	      ELSE
	        // Fehlerwiederholauftrag ??                   
	        IF #siErrorCount = #siMaxErrCount THEN
	          
	          // Wiederholungsauftrag wieder zurücknehmen
	          #sbWrStart2 := False;
	          #sbRdStart2 := False;
	          #sbWrite := False;
	          
	          //Fehlerzähler zurücksetzen
	          #siErrorCount := 0;
	          
	          
	          // Fehler ausgeben 
	          #sbError := #sbRdError;
	          
	          // nix tun bis Zähler überläuft
	        ELSE
	          #siErrorCount := #siErrorCount + 1;
	        END_IF;
	      END_IF;
	      
	      // Fehler : die Auftragsreferenz der Antwort übertimmt nicht mit der Auftragsreferenz der Anfrage überein
	    ELSIF NOT (#siReqRef = BYTE_TO_INT(#sxRespParaMulti.sxHeader.syReqRef)) AND NOT #sbRdBusy AND #pbValidSFB THEN
	      #siErrorId := 1;
	      #sbError := True;
	      #sbDone := False;
	      
	      // Wiederholungsauftrag wieder zurücknehmen
	      #sbWrStart2 := False;
	      #sbRdStart2 := False;
	      #sbWrite := False;
	      
	      // Fehler : falsche Auftragskennung zurück erhalten    
	    ELSIF NOT (#sxRespParaMulti.sxHeader.syReqId = B#16#82 OR #sxRespParaMulti.sxHeader.syReqId = B#16#02) AND
	      NOT #sbRdBusy AND #pbValidSFB THEN
	      #siErrorId := 1;
	      #sbError := True;
	      #sbDone := False;
	      
	      // Wiederholungsauftrag wieder zurücknehmen
	      #sbWrStart2 := False;
	      #sbRdStart2 := False;
	      #sbWrite := False;
	      
	      // Fehler : die angeforderte Anzahl Parameter entspricht nicht der übermittelten Anzahl Parameter überein
	    ELSIF NOT (#sxRespParaMulti.sxHeader.syParaNo = B#16#01) AND NOT #sbRdBusy AND #pbValidSFB THEN
	      #siErrorId := 1;
	      #sbError := True;
	      #sbDone := False;
	      
	      // Wiederholungsauftrag wieder zurücknehmen
	      #sbWrStart2 := False;
	      #sbRdStart2 := False;
	      #sbWrite := False;
	      
	      // Fehler : die Achse entspricht nicht der übergebenen Achse
	    ELSIF NOT (#syAxisNo = #sxRespParaMulti.sxHeader.syAxisNo) AND NOT #sbRdBusy AND #pbValidSFB THEN
	      #siErrorId := 1;
	      #sbError := True;
	      #sbDone := False;
	      
	      // Wiederholungsauftrag wieder zurücknehmen
	      #sbWrStart2 := False;
	      #sbRdStart2 := False;
	      #sbWrite := False;
	      
	      // kein Fehler beim LESEN AZYKLISCH und Auftrag fertig 
	    ELSIF NOT #sbRdBusy AND #pbValidSFB THEN
	      
	      // 2. Teilauftrag "Parameter schreiben bzw. ändern" negative Rückmeldung erhalten 
	      IF #sxRespParaMulti.sxHeader.syReqId = B#16#82 THEN
	        
	        // die angefragten Parameter auswerten und im Puffer abspeichern
	        // Format des Parameters auswerten, bei Format = Error Fehler auswerten 
	        IF (BYTE_TO_INT(#sxRespParaMulti.sxData[1]) = 68) THEN
	          
	          // Fehlerwert ermitteln und abspeichern 
	          // Format = Word, zwei Bytes zu übermitteltem Parameterwert zusammenfassen
	          #pwWordHigh := SHL(IN := BYTE_TO_WORD(#sxRespParaMulti.sxData[3]), N := 8);
	          #pwWordLow := BYTE_TO_WORD(#sxRespParaMulti.sxData[4]);
	          #pwWord1 := #pwWordHigh XOR #pwWordLow;
	            
	          #sbError := True;
	            
	          // ermittelte Fehlernummer im Puffer zurücksetzen
	          #ErrorNo := W#16#00;
	          
	          #ErrorNo := #pwWord1;
	          
	          // Die Fehlerhaftigkeit des erkannten Parameter in der Fehlernummer eintragen   
	          #swParaError := #swParaError OR W#16#01;
	          
	        ELSE
	          
	          // Die Fehlerhaftigkeit des erkannten Parameter in der Fehlernummer löschen   
	          #swParaError := #swParaError AND W#16#FFFE;
	          
	          // ermittelte Fehlernummer im Puffer zurücksetzen
	          #ErrorNo := W#16#00;
	        END_IF;
	      END_IF; // 2. Teilauftrag "Parameter schreiben bzw. ändern" negative Rückmeldung erhalten
	      
	      // Fehlerkennung zurücknehmen
	      IF (#siErrorId = 3) OR (#siErrorId = 1) THEN
	        #siErrorId := 0;
	        #sbError := False;
	      END_IF;
	      
	      #DiagId := W#16#00;
	      
	      // 2. Teilauftrag "Parameter schreiben bzw. ändern" ist abgeschlossen
	      #sbRdStart2 := False;
	      #sbWrite := False;
	      
	    END_IF; // kein Fehler beim LESEN AZYKLISCH und Auftrag fertig 
	  END_IF; // vom 2. Teilauftrag "Parameter schreiben bzw. ändern" die Antwort abwarten und dann auswerten 
	END_IF; // Auftrag "Parameter schreiben" wurde ausgelöst
	
	#pdDWordHigh := SHL(IN := INT_TO_DWORD(#siErrorId), N := 16);
	#pdDWordLow := WORD_TO_DWORD(#swParaError);
	
	// ermittelter Parameterwert eintragen (Word)
	#ErrorId := #pdDWordHigh XOR #pdDWordLow;
	
	// Initialisierung von Ausgängen
	#Busy := #sbBusy;
	#Error := #sbError;
	#Format := #syFormat;
	// Änderung wegen verhalten von Ready  
	#Done := #sbDone;
	// Prüfen, ob Auftrag abgeschlossen ist
	IF ((#Error OR #Done) AND NOT #sbReady) THEN
	  #Ready := True;
	  #sbReady := True;
	ELSE
	  #Ready := False;
	END_IF;
	
	
END_FUNCTION_BLOCK

FUNCTION_BLOCK "SINA_SPEED"
TITLE = 'Speed Control with SINAMICS and S7'
{ S7_Optimized_Access := 'TRUE' }
AUTHOR : DRVDPS7
FAMILY : DRIVES
NAME : SINA_SPD
VERSION : 5.1
//Copyright (C) Siemens AG 2012. All Rights Reserved. Confidential
//-------------------------------------------------------------------------------------- 
//SINA_SPEED: Drehzahlregelung mit dem Antriebsbaustein SINAMICS S120/G120 <-> S7-1200
//------------------------------------------------------------------------------------- Ersteller: Siemens AG Erlangen A&D MC PM   Datum:  07.07.10        Vers.:2.1
//Änderung:  J.B. Typical Team                       07.12.12              2.2
//    Umsetzung in SCL / TIA 
//Änderung:  J.B. Typical Team                       29.04.13              2.3
//    1. "Q" an den AusgÃ¤nge entfernen
//    2. Neuer Ausgang PwrInhibit
//Änderung:  J.B. Typical Team                       28.06.13              2.4
//    Ã„nderung HW-Zugriff Ã¼ber LOG2MOD
//     
//Änderung:  J.B. Typical Team                       18.07.13              2.5
//    Ã„nderung HW-Zugriff Ã¼ber zwei HW-EingÃ¤nge
//
//Änderung:  J.B. Typical Team                       17.07.14              3.0
//    Optimmierung
//
//Änderung:  J.B. Typical Team                       30.07.14              4.0
//    Festlegung auf einheitlicher neuer Version 4.0
//
//Änderung:  P.Z. Typical Team                       03.12.15              4.1
//    Schnittstelle an Programmierleitfadeb TIA-Potal angepasst
//    zusÃ¤tzlicher Eingang "ConfigAxis" fÃ¼r STW-Bits
//
//Änderung:  G.F. Typical Team                       01.03.16              4.2
//    Sollwert auf INT - Grenzen begrenzt
//Änderung:  F.G. Typical Team                       13.09.16              4.3
//    Ausgabewerte am Ausgang "Status" angepasst 
//
//Änderung:  G.F. Typical Team                       11.01.17              5.0
//    - Festlegung auf einheitlicher neuer Version 5.0 
//
//Änderung:  G.F. Typical Team                       03.05.18              5.1
//    - Alle Bits des Eingang ConfigAxis auf STW1 aufgelegt 
//
//Bibliothek V7
//Funktion: Drehzahlregelung mit dem Antriebsbaustein SINAMICS S120/G120 <-> S7-1200
//********************************************************************************************************************************************************
//************************************************************************FB283***************************************************************************
//********************************************************************************************************************************************************
   VAR_INPUT 
      EnableAxis : Bool := 0;   // 0-->1; 1 = Enable the drive (OFF2 / OFF 3 are 1 in default status) (OFF1 = 0-->1)
      AckError : Bool := 0;   // 1 = Acknowledge drive error
      SpeedSp : Real := 0.0;   // Speed standardises with the standardisation factor
      RefSpeed : Real := 0.0;   // Standardisation factor of speed
      ConfigAxis : Word := 16#003F;   // binary programmed input to control all functions in the telegram without its own function block input
      HWIDSTW : HW_IO := 0;   // Hardware Identifer set point slot
      HWIDZSW : HW_IO := 0;   // Hardware Identifer actual value slot
   END_VAR

   VAR_OUTPUT 
      AxisEnabled : Bool := 0;   // 1 = Drive is enabled
      Lockout : Bool := 0;   // 1 = Drive lockout active
      ActVelocity : Real := 0.0;   // Actual in [U/min]
      Error : Bool := 0;   // 1 = Error  (FB and Infeed)
      Status : Word := 0;   // Status output (7002 = FB in operation; 8xxx = error description  - read the manual)
      DiagId : Word := 16#0000;   // Error codes of the cyclic system funtion blocks DPWR / DPRD_DAT
   END_VAR

   VAR 
      sxSendBuf : Struct   // Send buffer
         STW1 : Word := WORD#16#0000;   // STW1sxSTW1     : STRUCT            Bit08       : BOOL:=False;              // ST-Wort-1 Bit 08 --> Reserve            Bit09       : BOOL:=False;              // ST-Wort-1 Bit 09 --> Reserve            Bit10       : BOOL:=True;               // ST-Wort-1 Bit 10 --> FÃ¼hrung durch PLC            Dir         : BOOL:=False;              // ST-Wort-1 Bit 11 --> Direction            Bit12       : BOOL:=False;              // ST-Wort-1 Bit 12 --> Haltebremse unbedingt Ã¶ffnen            Bit13       : BOOL:=False;              // ST-Wort-1 Bit 13 --> Motorpotenziometer Sollwert hÃ¶her            Bit14       : BOOL:=False;              // ST-Wort-1 Bit 14 --> Motorpotenziometer Sollwert tiefer            Bit15       : BOOL:=False;              // ST-Wort-1 Bit 15 --> Reserviert            Off1        : BOOL:=False;              // ST-Wort-1 Bit 00 --> OFF1/ON (flanks acceptance)            Off2        : BOOL:=True;               // ST-Wort-1 Bit 01 --> OFF2/ON (enable possible)            Off3        : BOOL:=True;               // ST-Wort-1 Bit 02 --> OFF3/ON (enable possible)            InvEn       : BOOL:=True;               // ST-Wort-1 Bit 03 --> Enable controller            RampEn      : BOOL:=True;               // ST-Wort-1 Bit 04 --> Ramp enable            RampOn      : BOOL:=True;               // ST-Wort-1 Bit 05 --> Ramp On            SpEn        : BOOL:=True;               // ST-Wort-1 Bit 06 --> Speed set point enable            AckFlt      : BOOL:=False;              // ST-Wort-1 Bit 07 --> Acknowledge fault         END_STRUCT;
         Velocity : Word := WORD#16#0000;   // Setpoint of velocity
      END_STRUCT;
      sxRecvBuf : Struct   // Receive buffer
         ZSW1 : Word := WORD#16#0000;   // ZSW1sxZSW1     : STRUCT            SpDev       : BOOL:=False;              // ZSW-Wort-1 = Schleppfehler im Toleranzbereich            Pcd         : BOOL:=False;              // ZSW-Wort-1 = PZD-FÃ¼hrung erreicht            Comp        : BOOL:=False;              // ZSW-Wort-1 = Zielposition erreicht            CurLim      : BOOL:=False;              // ZSW-Wort-1 = Referenzpunkt gesetzt            Brake       : BOOL:=False;              // ZSW-Wort-1 = Haltebremse Ã¶ffnen            Motover     : BOOL:=False;              // ZSW-Wort-1 = keine Warnung Ãœbertemperatur Motor            Dir         : BOOL:=False;              // ZSW-Wort-1 = Direction            Invover     : BOOL:=False;              // ZSW-Wort-1 = keine Warnung thermische Ãœberlast Leistungsteil            Rts         : BOOL:=False;              // ZSW-Wort-1 = Ready to power up / to start            Rdy         : BOOL:=False;              // ZSW-Wort-1 = Ready to operate            IOp         : BOOL:=False;              // ZSW-Wort-1 = In operation (operation enabled)            Fault       : BOOL:=False;              // ZSW-Wort-1 = Fault present            NoOff2      : BOOL:=False;              // ZSW-Wort-1 = OFF2 inactive            NoOff3      : BOOL:=False;              // ZSW-Wort-1 = OFF3 inactive            Inhibit     : BOOL:=False;              // ZSW-Wort-1 = Power ON inhibit active             Alarm       : BOOL:=False;              // ZSW-Wort-1 = Alarm / Warning present                     END_STRUCT;
         Velocity : Word := WORD#16#0000;   // Feedback of velocity
      END_STRUCT;
   END_VAR

   VAR_TEMP 
      piRetSFC : Int;   // Status for fault analysis
      piCount : Int;   // Freely available counter variable 3
      prVelocity : Real;   // velocity
      pdRecvBuf : DWord;   // Buffer of Recv-Value
      pdSendBuf : DWord;   // Buffer of Send-Value
      phLAddr : HW_IO;   // Start addr from the I/O process image area of mod (DEC) for DPWR_DAT/DPRD_DAT
      swSendBuf : Array[0..1] of Word;   // Sendepuffer
      swRecvBuf : Array[0..1] of Word;   // Empfangspuffer         Static variables
   END_VAR


BEGIN
	
	//=============================================================================
	//SIEMENS AG
	//(c)Copyright 2017 All Rights Reserved
	//-----------------------------------------------------------------------------
	// Library: DriveLib
	// Tested with: S7-1516-3 PN/DP V1.8
	// Engineering: TIA Portal V14
	// Restrictions: -
	// Requirements: S7-1200 / S7-1500
	// Functionality: cyclic communication between a SINAMICS a PLC.
	//                If in HWConfig Std.TLG 1 is projected 2 PZD-words are exchanged
	//                in every bus cycle.
	//                The parametrisation of these words is described in the manual of the
	//                SINAMICS
	//=============================================================================
	
	// Schreibdaten zusammenstellen
	// Steuerword aufbereiten
	
	#sxSendBuf.STW1.%X0 := #EnableAxis;
	#sxSendBuf.STW1.%X1 := #ConfigAxis.%X0;
	#sxSendBuf.STW1.%X2 := #ConfigAxis.%X1;
	#sxSendBuf.STW1.%X3 := #ConfigAxis.%X2;
	#sxSendBuf.STW1.%X4 := #ConfigAxis.%X3;
	#sxSendBuf.STW1.%X5 := #ConfigAxis.%X4;
	#sxSendBuf.STW1.%X6 := #ConfigAxis.%X5;
	#sxSendBuf.STW1.%X7 := #AckError;
	#sxSendBuf.STW1.%X8 := #ConfigAxis.%X10;
	#sxSendBuf.STW1.%X9 := #ConfigAxis.%X11;
	#sxSendBuf.STW1.%X10 := TRUE;
	#sxSendBuf.STW1.%X11 := #ConfigAxis.%X6;
	#sxSendBuf.STW1.%X12 := #ConfigAxis.%X7;
	#sxSendBuf.STW1.%X13 := #ConfigAxis.%X8;
	#sxSendBuf.STW1.%X14 := #ConfigAxis.%X9;
	#sxSendBuf.STW1.%X15 := #ConfigAxis.%X12;
	
	// Geschwindigkeit
	IF #RefSpeed <> 0 THEN
	  #prVelocity := #SpeedSp * (16384.0 / #RefSpeed);
	  // Limit REAL - Variable to INT - Limits
	  IF #prVelocity > 32767 THEN
	    #prVelocity := 32767;
	  ELSIF #prVelocity < -32768 THEN
	    #prVelocity := -32768;
	  ELSE
	    ; // not needed
	  END_IF;
	  #sxSendBuf.Velocity := INT_TO_WORD(REAL_TO_INT(#prVelocity));
	  
	ELSE
	  #sxSendBuf.Velocity := W#16#0;
	END_IF;
	#swSendBuf[0] := #sxSendBuf.STW1;
	#swSendBuf[1] := #sxSendBuf.Velocity;
	
	//Prozessdaten zur Signalbaugruppe schreiben
	#piRetSFC := DPWR_DAT(LADDR := #HWIDSTW,
	                      RECORD := #swSendBuf);
	
	// Fehler der RÃ¼ckmeldung ausgeben
	#DiagId := INT_TO_WORD(#piRetSFC);
	
	//kein Fehler beim Schreiben
	IF #piRetSFC = 0 THEN
	  
	  //kein Fehler beim Schreiben
	  IF #piRetSFC = 0 THEN
	    
	    //Prozessdaten von der Signalbaugruppe lesen
	    #piRetSFC := DPRD_DAT(LADDR := #HWIDZSW,
	                          RECORD => #swRecvBuf);
	    
	    // Fehler der RÃ¼ckmeldung ausgeben
	    #DiagId := INT_TO_WORD(#piRetSFC);
	  END_IF;
	  
	  //Fehler beim Lesen (Profibus-Kommunikation unterbrochen)
	  IF #piRetSFC <> 0 THEN
	    
	    // Fehler
	    #Error := TRUE;
	    #Status := 16#8600;
	    
	    // Zustandsworte lÃ¶schen
	    #sxRecvBuf.ZSW1.%X8 := 0;
	    #sxRecvBuf.ZSW1.%X9 := 0;
	    #sxRecvBuf.ZSW1.%X10 := 0;
	    #sxRecvBuf.ZSW1.%X11 := 0;
	    #sxRecvBuf.ZSW1.%X12 := 0;
	    #sxRecvBuf.ZSW1.%X13 := 0;
	    #sxRecvBuf.ZSW1.%X14 := 0;
	    #sxRecvBuf.ZSW1.%X15 := 0;
	    #sxRecvBuf.ZSW1.%X0 := 0;
	    #sxRecvBuf.ZSW1.%X1 := 0;
	    #sxRecvBuf.ZSW1.%X2 := 0;
	    #sxRecvBuf.ZSW1.%X3 := 0;
	    #sxRecvBuf.ZSW1.%X4 := 0;
	    #sxRecvBuf.ZSW1.%X5 := 0;
	    #sxRecvBuf.ZSW1.%X6 := 0;
	    #sxRecvBuf.ZSW1.%X7 := 0;
	    
	    
	    (*#sxRecvBuf.sxZSW1.SpDev   := 0;
	    #sxRecvBuf.sxZSW1.Pcd     := 0;
	    #sxRecvBuf.sxZSW1.Comp    := 0;
	    #sxRecvBuf.sxZSW1.CurLim  := 0;
	    #sxRecvBuf.sxZSW1.Brake   := 0;
	    #sxRecvBuf.sxZSW1.Motover := 0;
	    #sxRecvBuf.sxZSW1.Dir     := 0;
	    #sxRecvBuf.sxZSW1.Invover := 0;
	    #sxRecvBuf.sxZSW1.Rts     := 0;
	    #sxRecvBuf.sxZSW1.Rdy     := 0;
	    #sxRecvBuf.sxZSW1.IOp     := 0;
	    #sxRecvBuf.sxZSW1.Fault   := 0;
	    #sxRecvBuf.sxZSW1.NoOff2  := 0;
	    #sxRecvBuf.sxZSW1.NoOff3  := 0;
	    #sxRecvBuf.sxZSW1.Inhibit := 0;
	    #sxRecvBuf.sxZSW1.Alarm   := 0;*)
	    
	    #sxRecvBuf.Velocity := W#16#00;
	    
	    // Werte auslesen
	  ELSE
	    #sxRecvBuf.ZSW1 := #swRecvBuf[0];
	    #sxRecvBuf.Velocity := #swRecvBuf[1];
	    
	    // ZSW1 aufbereiten                       
	    #AxisEnabled := #sxRecvBuf.ZSW1.%X2;
	    #Error := #sxRecvBuf.ZSW1.%X3 OR #sxRecvBuf.ZSW1.%X6;
	    #Lockout := #sxRecvBuf.ZSW1.%X6;
	    
	    // Fehler auswerten
	    IF #sxRecvBuf.ZSW1.%X3 THEN
	      #Status := 16#8401;
	    ELSIF #sxRecvBuf.ZSW1.%X6 THEN
	      #Status := 16#8402;
	    ELSE
	      #Status := 16#7002;
	    END_IF;
	    
	    (*#Busy       := #sxRecvBuf.sxZSW1.IOp;
	    #Error      := #sxRecvBuf.sxZSW1.Fault OR #sxRecvBuf.sxZSW1.Inhibit;
	    #PwrInhibit := #sxRecvBuf.sxZSW1.Inhibit;            
	
	    // Fehler auswerten
	    IF #sxRecvBuf.sxZSW1.Fault THEN
	        #ErrorId := 1;
	    ELSIF #sxRecvBuf.sxZSW1.Inhibit THEN 
	        #ErrorId := 2;
	    ELSE
	        #ErrorId := 0;    
	    END_IF;*)
	    
	    // Geschwindigkeit
	    IF #RefSpeed <> 0 THEN
	      #ActVelocity := INT_TO_REAL(WORD_TO_INT(#sxRecvBuf.Velocity)) / (16384.0 / #RefSpeed);
	    ELSE
	      #ActVelocity := 0.0;
	    END_IF;
	  END_IF;
	ELSE
	  
	  // Fehler
	  #Error := TRUE;
	  #Status := 16#8601;
	  
	END_IF;
	
	
	
END_FUNCTION_BLOCK

DATA_BLOCK "Obj_St1"   // DB100
VERSION : 0.1
// stored: AutoNumber false, DBAccessibleFromOPCUA true, DBAccessibleFromWebserver true, InstanceOfName Obj_St1_FB, InstanceOfType FB
"Obj_St1_FB"
BEGIN
END_DATA_BLOCK

DATA_BLOCK "Obj_St2"   // DB200
VERSION : 0.1
// stored: AutoNumber false, DBAccessibleFromOPCUA true, DBAccessibleFromWebserver true, InstanceOfName Obj_St2_FB, InstanceOfType FB
"Obj_St2_FB"
BEGIN
END_DATA_BLOCK

DATA_BLOCK "Obj_St3"   // DB300
VERSION : 0.1
// stored: AutoNumber false, DBAccessibleFromOPCUA true, DBAccessibleFromWebserver true, InstanceOfName Obj_St3_FB, InstanceOfType FB
"Obj_St3_FB"
BEGIN
END_DATA_BLOCK

DATA_BLOCK "Obj_St4"   // DB400
VERSION : 0.1
// stored: AutoNumber false, DBAccessibleFromOPCUA true, DBAccessibleFromWebserver true, InstanceOfName Obj_St4_FB, InstanceOfType FB
"Obj_St4_FB"
BEGIN
END_DATA_BLOCK

DATA_BLOCK "Cfg_St1_Axe_X"   // DB170
AUTHOR : DRVDPS7
FAMILY : DRIVES
NAME : SINA_POS
VERSION : 5.7
// stored: AutoNumber false, DBAccessibleFromOPCUA true, DBAccessibleFromWebserver true, InstanceOfName SINA_POS, InstanceOfType FB
"SINA_POS"
BEGIN
END_DATA_BLOCK

DATA_BLOCK "Cfg_St1_Axe_Y"   // DB175
AUTHOR : DRVDPS7
FAMILY : DRIVES
NAME : SINA_POS
VERSION : 5.7
// stored: AutoNumber false, DBAccessibleFromOPCUA true, DBAccessibleFromWebserver true, InstanceOfName SINA_POS, InstanceOfType FB
"SINA_POS"
BEGIN
END_DATA_BLOCK

DATA_BLOCK "Cfg_St1_Prehenseur_Z"   // DB180
AUTHOR : DRVDPS7
FAMILY : DRIVES
NAME : SINA_POS
VERSION : 5.7
// stored: AutoNumber false, DBAccessibleFromOPCUA true, DBAccessibleFromWebserver true, InstanceOfName SINA_POS, InstanceOfType FB
"SINA_POS"
BEGIN
END_DATA_BLOCK

DATA_BLOCK "G7A_St1_Init"   // DB110
VERSION : 0.1
// stored: AutoNumber false, DBAccessibleFromOPCUA true, DBAccessibleFromWebserver true, InstanceOfName G7A_St1_Init_FB, InstanceOfType FB
"G7A_St1_Init_FB"
BEGIN
END_DATA_BLOCK

DATA_BLOCK "G7A_St1_Start"   // DB120
VERSION : 0.1
// stored: AutoNumber false, DBAccessibleFromOPCUA true, DBAccessibleFromWebserver true, InstanceOfName G7A_St1_Start_FB, InstanceOfType FB
"G7A_St1_Start_FB"
BEGIN
END_DATA_BLOCK

DATA_BLOCK "G7A_St1_Execute"   // DB130
VERSION : 0.1
// stored: AutoNumber false, DBAccessibleFromOPCUA true, DBAccessibleFromWebserver true, InstanceOfName G7A_St1_Execute_FB, InstanceOfType FB
"G7A_St1_Execute_FB"
BEGIN
END_DATA_BLOCK

DATA_BLOCK "G7A_St1_End"   // DB140
VERSION : 0.1
// stored: AutoNumber false, DBAccessibleFromOPCUA true, DBAccessibleFromWebserver true, InstanceOfName G7A_St1_End_FB, InstanceOfType FB
"G7A_St1_End_FB"
BEGIN
END_DATA_BLOCK

DATA_BLOCK "G7A_St1_Stop"   // DB150
VERSION : 0.1
// stored: AutoNumber false, DBAccessibleFromOPCUA true, DBAccessibleFromWebserver true, InstanceOfName G7A_St1_Stop_FB, InstanceOfType FB
"G7A_St1_Stop_FB"
BEGIN
END_DATA_BLOCK

DATA_BLOCK "Cfg_St2_Axe_X1"   // DB270
AUTHOR : DRVDPS7
FAMILY : DRIVES
NAME : SINA_POS
VERSION : 5.7
// stored: AutoNumber false, DBAccessibleFromOPCUA true, DBAccessibleFromWebserver true, InstanceOfName SINA_POS, InstanceOfType FB
"SINA_POS"
BEGIN
END_DATA_BLOCK

DATA_BLOCK "Cfg_St2_Axe_X2"   // DB275
AUTHOR : DRVDPS7
FAMILY : DRIVES
NAME : SINA_POS
VERSION : 5.7
// stored: AutoNumber false, DBAccessibleFromOPCUA true, DBAccessibleFromWebserver true, InstanceOfName SINA_POS, InstanceOfType FB
"SINA_POS"
BEGIN
END_DATA_BLOCK

DATA_BLOCK "Cfg_St2_Prehenseur_Z"   // DB280
AUTHOR : DRVDPS7
FAMILY : DRIVES
NAME : SINA_POS
VERSION : 5.7
// stored: AutoNumber false, DBAccessibleFromOPCUA true, DBAccessibleFromWebserver true, InstanceOfName SINA_POS, InstanceOfType FB
"SINA_POS"
BEGIN
END_DATA_BLOCK

DATA_BLOCK "G7A_St2_Init"   // DB210
VERSION : 0.1
// stored: AutoNumber false, DBAccessibleFromOPCUA true, DBAccessibleFromWebserver true, InstanceOfName G7A_St2_Init_FB, InstanceOfType FB
"G7A_St2_Init_FB"
BEGIN
END_DATA_BLOCK

DATA_BLOCK "G7A_St2_Start"   // DB220
VERSION : 0.1
// stored: AutoNumber false, DBAccessibleFromOPCUA true, DBAccessibleFromWebserver true, InstanceOfName G7A_St2_Start_FB, InstanceOfType FB
"G7A_St2_Start_FB"
BEGIN
END_DATA_BLOCK

DATA_BLOCK "G7A_St2_Execute"   // DB230
VERSION : 0.1
// stored: AutoNumber false, DBAccessibleFromOPCUA true, DBAccessibleFromWebserver true, InstanceOfName G7A_St2_Execute_FB, InstanceOfType FB
"G7A_St2_Execute_FB"
BEGIN
END_DATA_BLOCK

DATA_BLOCK "G7A_St2_End"   // DB240
VERSION : 0.1
// stored: AutoNumber false, DBAccessibleFromOPCUA true, DBAccessibleFromWebserver true, InstanceOfName G7A_St2_End_FB, InstanceOfType FB
"G7A_St2_End_FB"
BEGIN
END_DATA_BLOCK

DATA_BLOCK "G7A_St2_Stop"   // DB250
VERSION : 0.1
// stored: AutoNumber false, DBAccessibleFromOPCUA true, DBAccessibleFromWebserver true, InstanceOfName G7A_St2_Stop_FB, InstanceOfType FB
"G7A_St2_Stop_FB"
BEGIN
END_DATA_BLOCK

DATA_BLOCK "Cfg_St3_Axe_X1"   // DB370
AUTHOR : DRVDPS7
FAMILY : DRIVES
NAME : SINA_POS
VERSION : 5.7
// stored: AutoNumber false, DBAccessibleFromOPCUA true, DBAccessibleFromWebserver true, InstanceOfName SINA_POS, InstanceOfType FB
"SINA_POS"
BEGIN
END_DATA_BLOCK

DATA_BLOCK "Cfg_St3_Axe_X2"   // DB375
AUTHOR : DRVDPS7
FAMILY : DRIVES
NAME : SINA_POS
VERSION : 5.7
// stored: AutoNumber false, DBAccessibleFromOPCUA true, DBAccessibleFromWebserver true, InstanceOfName SINA_POS, InstanceOfType FB
"SINA_POS"
BEGIN
END_DATA_BLOCK

DATA_BLOCK "Cfg_St3_Axe_Y"   // DB380
AUTHOR : DRVDPS7
FAMILY : DRIVES
NAME : SINA_POS
VERSION : 5.7
// stored: AutoNumber false, DBAccessibleFromOPCUA true, DBAccessibleFromWebserver true, InstanceOfName SINA_POS, InstanceOfType FB
"SINA_POS"
BEGIN
END_DATA_BLOCK

DATA_BLOCK "Cfg_St3_Axe_Z"   // DB385
AUTHOR : DRVDPS7
FAMILY : DRIVES
NAME : SINA_POS
VERSION : 5.7
// stored: AutoNumber false, DBAccessibleFromOPCUA true, DBAccessibleFromWebserver true, InstanceOfName SINA_POS, InstanceOfType FB
"SINA_POS"
BEGIN
END_DATA_BLOCK

DATA_BLOCK "G7A_St3_Init"   // DB310
VERSION : 0.1
// stored: AutoNumber false, DBAccessibleFromOPCUA true, DBAccessibleFromWebserver true, InstanceOfName G7A_St3_Init_FB, InstanceOfType FB
"G7A_St3_Init_FB"
BEGIN
END_DATA_BLOCK

DATA_BLOCK "G7A_St3_Start"   // DB320
VERSION : 0.1
// stored: AutoNumber false, DBAccessibleFromOPCUA true, DBAccessibleFromWebserver true, InstanceOfName G7A_St3_Start_FB, InstanceOfType FB
"G7A_St3_Start_FB"
BEGIN
END_DATA_BLOCK

DATA_BLOCK "G7A_St3_Execute"   // DB330
VERSION : 0.1
// stored: AutoNumber false, DBAccessibleFromOPCUA true, DBAccessibleFromWebserver true, InstanceOfName G7A_St3_Execute_FB, InstanceOfType FB
"G7A_St3_Execute_FB"
BEGIN
END_DATA_BLOCK

DATA_BLOCK "G7A_St3_End"   // DB340
VERSION : 0.1
// stored: AutoNumber false, DBAccessibleFromOPCUA true, DBAccessibleFromWebserver true, InstanceOfName G7A_St3_End_FB, InstanceOfType FB
"G7A_St3_End_FB"
BEGIN
END_DATA_BLOCK

DATA_BLOCK "G7A_St3_Stop"   // DB350
VERSION : 0.1
// stored: AutoNumber false, DBAccessibleFromOPCUA true, DBAccessibleFromWebserver true, InstanceOfName G7A_St3_Stop_FB, InstanceOfType FB
"G7A_St3_Stop_FB"
BEGIN
END_DATA_BLOCK

DATA_BLOCK "Cfg_St4_Axe_X1"   // DB475
AUTHOR : DRVDPS7
FAMILY : DRIVES
NAME : SINA_POS
VERSION : 5.7
// stored: AutoNumber false, DBAccessibleFromOPCUA true, DBAccessibleFromWebserver true, InstanceOfName SINA_POS, InstanceOfType FB
"SINA_POS"
BEGIN
END_DATA_BLOCK

DATA_BLOCK "Cfg_St4_Axe_Y1"   // DB480
AUTHOR : DRVDPS7
FAMILY : DRIVES
NAME : SINA_POS
VERSION : 5.7
// stored: AutoNumber false, DBAccessibleFromOPCUA true, DBAccessibleFromWebserver true, InstanceOfName SINA_POS, InstanceOfType FB
"SINA_POS"
BEGIN
END_DATA_BLOCK

DATA_BLOCK "Cfg_St4_Axe_Y2"   // DB485
AUTHOR : DRVDPS7
FAMILY : DRIVES
NAME : SINA_POS
VERSION : 5.7
// stored: AutoNumber false, DBAccessibleFromOPCUA true, DBAccessibleFromWebserver true, InstanceOfName SINA_POS, InstanceOfType FB
"SINA_POS"
BEGIN
END_DATA_BLOCK

DATA_BLOCK "Cfg_St4_Prehenseur_Z2"   // DB490
AUTHOR : DRVDPS7
FAMILY : DRIVES
NAME : SINA_POS
VERSION : 5.7
// stored: AutoNumber false, DBAccessibleFromOPCUA true, DBAccessibleFromWebserver true, InstanceOfName SINA_POS, InstanceOfType FB
"SINA_POS"
BEGIN
END_DATA_BLOCK

DATA_BLOCK "Cfg_St4_Prehenseur_Z3"   // DB495
AUTHOR : DRVDPS7
FAMILY : DRIVES
NAME : SINA_POS
VERSION : 5.7
// stored: AutoNumber false, DBAccessibleFromOPCUA true, DBAccessibleFromWebserver true, InstanceOfName SINA_POS, InstanceOfType FB
"SINA_POS"
BEGIN
END_DATA_BLOCK

DATA_BLOCK "G7A_St4_Init"   // DB410
VERSION : 0.1
// stored: AutoNumber false, DBAccessibleFromOPCUA true, DBAccessibleFromWebserver true, InstanceOfName G7A_St4_Init_FB, InstanceOfType FB
"G7A_St4_Init_FB"
BEGIN
END_DATA_BLOCK

DATA_BLOCK "G7A_St4_Start"   // DB420
VERSION : 0.1
// stored: AutoNumber false, DBAccessibleFromOPCUA true, DBAccessibleFromWebserver true, InstanceOfName G7A_St4_Start_FB, InstanceOfType FB
"G7A_St4_Start_FB"
BEGIN
END_DATA_BLOCK

DATA_BLOCK "G7A_St4.1_Execute"   // DB430
VERSION : 0.1
// stored: AutoNumber false, DBAccessibleFromOPCUA true, DBAccessibleFromWebserver true, InstanceOfName G7A_St4.1_Execute_FB, InstanceOfType FB
"G7A_St4.1_Execute_FB"
BEGIN
END_DATA_BLOCK

DATA_BLOCK "G7A_St4.2_Execute"   // DB440
VERSION : 0.1
// stored: AutoNumber false, DBAccessibleFromOPCUA true, DBAccessibleFromWebserver true, InstanceOfName G7A_St4.2_Execute_FB, InstanceOfType FB
"G7A_St4.2_Execute_FB"
BEGIN
END_DATA_BLOCK

DATA_BLOCK "G7A_St4.3_Execute"   // DB450
VERSION : 0.1
// stored: AutoNumber false, DBAccessibleFromOPCUA true, DBAccessibleFromWebserver true, InstanceOfName G7A_St4.3_Execute_FB, InstanceOfType FB
"G7A_St4.3_Execute_FB"
BEGIN
END_DATA_BLOCK

DATA_BLOCK "G7A_St4_End"   // DB460
VERSION : 0.1
// stored: AutoNumber false, DBAccessibleFromOPCUA true, DBAccessibleFromWebserver true, InstanceOfName G7A_St4_End_FB, InstanceOfType FB
"G7A_St4_End_FB"
BEGIN
END_DATA_BLOCK

DATA_BLOCK "G7A_St4_Stop"   // DB470
VERSION : 0.1
// stored: AutoNumber false, DBAccessibleFromOPCUA true, DBAccessibleFromWebserver true, InstanceOfName G7A_St4_Stop_FB, InstanceOfType FB
"G7A_St4_Stop_FB"
BEGIN
END_DATA_BLOCK

DATA_BLOCK "S00_Mode"   // DB1010
VERSION : 0.1
// stored: AutoNumber false, DBAccessibleFromOPCUA true, DBAccessibleFromWebserver true, InstanceOfName S00_Mode_FB, InstanceOfType FB
"S00_Mode_FB"
BEGIN
END_DATA_BLOCK

DATA_BLOCK "S10_Aborting"   // DB1020
VERSION : 0.1
// stored: AutoNumber false, DBAccessibleFromOPCUA true, DBAccessibleFromWebserver true, InstanceOfName S10_Aborting_FB, InstanceOfType FB
"S10_Aborting_FB"
BEGIN
END_DATA_BLOCK

DATA_BLOCK "S20_Aborted"   // DB1030
VERSION : 0.1
// stored: AutoNumber false, DBAccessibleFromOPCUA true, DBAccessibleFromWebserver true, InstanceOfName S20_Aborted_FB, InstanceOfType FB
"S20_Aborted_FB"
BEGIN
END_DATA_BLOCK

DATA_BLOCK "S30_Initializing"   // DB1040
VERSION : 0.1
// stored: AutoNumber false, DBAccessibleFromOPCUA true, DBAccessibleFromWebserver true, InstanceOfName S30_Initializing_FB, InstanceOfType FB
"S30_Initializing_FB"
BEGIN
END_DATA_BLOCK

DATA_BLOCK "S40_Acquitement"   // DB1050
VERSION : 0.1
// stored: AutoNumber false, DBAccessibleFromOPCUA true, DBAccessibleFromWebserver true, InstanceOfName S40_Acquitement_FB, InstanceOfType FB
"S40_Acquitement_FB"
BEGIN
END_DATA_BLOCK

DATA_BLOCK "S50_Ready"   // DB1060
VERSION : 0.1
// stored: AutoNumber false, DBAccessibleFromOPCUA true, DBAccessibleFromWebserver true, InstanceOfName S50_Ready_FB, InstanceOfType FB
"S50_Ready_FB"
BEGIN
END_DATA_BLOCK

DATA_BLOCK "S55_Ready_exit"   // DB1065
VERSION : 0.1
// stored: AutoNumber false, DBAccessibleFromOPCUA true, DBAccessibleFromWebserver true, InstanceOfName S55_Ready_exit_FB, InstanceOfType FB
"S55_Ready_exit_FB"
BEGIN
END_DATA_BLOCK

DATA_BLOCK "S60_Starting"   // DB1070
VERSION : 0.1
// stored: AutoNumber false, DBAccessibleFromOPCUA true, DBAccessibleFromWebserver true, InstanceOfName S60_Starting_FB, InstanceOfType FB
"S60_Starting_FB"
BEGIN
END_DATA_BLOCK

DATA_BLOCK "S70_Execute"   // DB1080
VERSION : 0.1
// stored: AutoNumber false, DBAccessibleFromOPCUA true, DBAccessibleFromWebserver true, InstanceOfName S70_Execute_FB, InstanceOfType FB
"S70_Execute_FB"
BEGIN
END_DATA_BLOCK

DATA_BLOCK "S80_End"   // DB1090
VERSION : 0.1
// stored: AutoNumber false, DBAccessibleFromOPCUA true, DBAccessibleFromWebserver true, InstanceOfName S80_End_FB, InstanceOfType FB
"S80_End_FB"
BEGIN
END_DATA_BLOCK

DATA_BLOCK "S90_Stopping"   // DB1100
VERSION : 0.1
// stored: AutoNumber false, DBAccessibleFromOPCUA true, DBAccessibleFromWebserver true, InstanceOfName S90_Stopping_FB, InstanceOfType FB
"S90_Stopping_FB"
BEGIN
END_DATA_BLOCK
